// TIA Portal V20 export
DATA_BLOCK "RealDbName"   // DB7
// Real comment mentioning RealSite.
   VAR
      RealFlag : Bool;
   END_VAR
   VAR RETAIN
      RealWord : Word := 16#0041;
   END_VAR
   VAR
      RealArray : Array[0..2] of Int;
      RealName : String := 'Real Site Name';
   END_VAR
BEGIN
END_DATA_BLOCK
